(* CoDeSys 2.3 export: FGETK16PUMP.EXP *)

(* POU K16/fGetK16Pump, ST *)
FUNCTION fGetK16Pump :BOOL
(* Проверка включения насоса*)
VAR_INPUT
	PumpID : USINT;
END_VAR
fGetK16Pump := PLC160DO.K16Pump[PumpID];
END_FUNCTION
